// TIA Portal project "start-start-start" (V16)

(* hardware
DEVICE "S7-1200 station_1"  S7-1200 Station
   slot 0: "Rack_0"  S7-1200 Rack  Rack  V1.0
   slot 1: "PLC_1"  CPU 1212C AC/DC/Rly  6ES7 212-1BE40-0XB0  V4.0
*)

// ===== PLC "PLC_1"  CPU 1212C AC/DC/Rly =====

VAR_GLOBAL   // PLC tag table "Default tag table"
   "start" AT %I0.1 : Bool;
   "stop" AT %I0.0 : Bool;
   "motor 1" AT %Q0.0 : Bool;
   "motor 2" AT %Q0.1 : Bool;
   "motor 3" AT %Q0.2 : Bool;
   "series Marker 1" AT %M0.0 : Bool;
   "Tag_1" AT %M0.1 : Bool;
   "Tag_2" AT %M0.3 : Bool;
   "Tag_3" AT %M0.4 : Bool;
   "series marker 2" AT %M0.5 : Bool;
   "Tag_4" AT %M0.6 : Bool;
END_VAR

ORGANIZATION_BLOCK "Main"   // OB1, LAD, ProgramCycle
TITLE = "Main Program Sweep (Cycle)"
{ S7_Optimized_Access := 'TRUE' }
VERSION : 0.1
   VAR_INPUT
      Initial_Call : Bool;   // Initial call of this OB
      Remanence : Bool;   // =True, if remanent data are available
   END_VAR
   VAR_TEMP   // added for the SCL form of the ladder/FBD networks
      _w1 : Bool;
   END_VAR
BEGIN

REGION Network 1
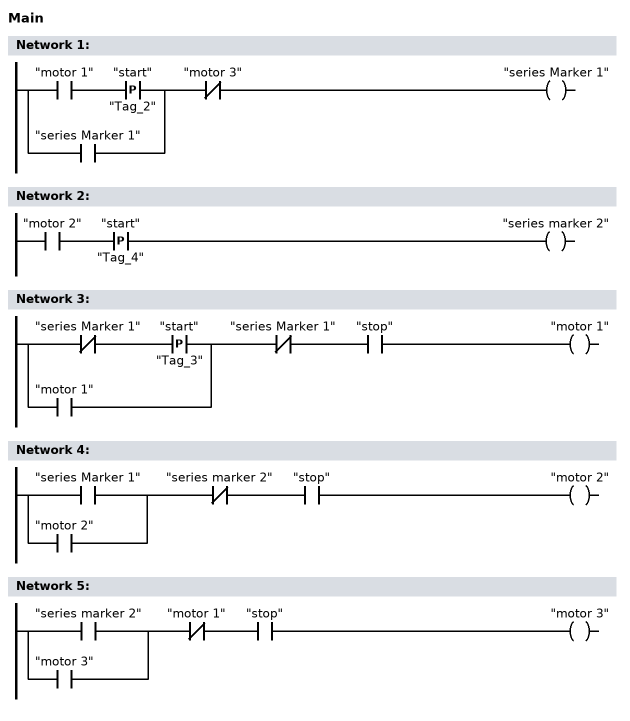
   RUNG wire#powerrail
      Contact( "motor 1" )
      P_Contact(operand := "start", bit := "Tag_2")
      wire#w1
      I_Contact( "motor 3" )
      Coil( "series Marker 1" )
   END_RUNG
   RUNG wire#powerrail
      Contact( "series Marker 1" )
   END_RUNG wire#w1
   // the same network as SCL:
   #_w1 := "motor 1" AND "start" AND NOT "Tag_2";   // rising edge of "start"
   "Tag_2" := "start";
   "series Marker 1" := (#_w1 OR "series Marker 1") AND NOT "motor 3";
END_REGION

REGION Network 2
   RUNG wire#powerrail
      Contact( "motor 2" )
      P_Contact(operand := "start", bit := "Tag_4")
      Coil( "series marker 2" )
   END_RUNG
   // the same network as SCL:
   #_w1 := "motor 2" AND "start" AND NOT "Tag_4";   // rising edge of "start"
   "Tag_4" := "start";
   "series marker 2" := #_w1;
END_REGION

REGION Network 3
   RUNG wire#powerrail
      I_Contact( "series Marker 1" )
      P_Contact(operand := "start", bit := "Tag_3")
      wire#w1
      I_Contact( "series Marker 1" )
      Contact( "stop" )
      Coil( "motor 1" )
   END_RUNG
   RUNG wire#powerrail
      Contact( "motor 1" )
   END_RUNG wire#w1
   // the same network as SCL:
   #_w1 := NOT "series Marker 1" AND "start" AND NOT "Tag_3";   // rising edge of "start"
   "Tag_3" := "start";
   "motor 1" := (#_w1 OR "motor 1") AND NOT "series Marker 1" AND "stop";
END_REGION

REGION Network 4
   RUNG wire#powerrail
      Contact( "series Marker 1" )
      wire#w1
      I_Contact( "series marker 2" )
      Contact( "stop" )
      Coil( "motor 2" )
   END_RUNG
   RUNG wire#powerrail
      Contact( "motor 2" )
   END_RUNG wire#w1
   // the same network as SCL:
   "motor 2" := ("series Marker 1" OR "motor 2") AND NOT "series marker 2" AND "stop";
END_REGION

REGION Network 5
   RUNG wire#powerrail
      Contact( "series marker 2" )
      wire#w1
      I_Contact( "motor 1" )
      Contact( "stop" )
      Coil( "motor 3" )
   END_RUNG
   RUNG wire#powerrail
      Contact( "motor 3" )
   END_RUNG wire#w1
   // the same network as SCL:
   "motor 3" := ("series marker 2" OR "motor 3") AND NOT "motor 1" AND "stop";
END_REGION
END_ORGANIZATION_BLOCK